FUNCTION alg_g_a_X2: LREAL
{ S7_Optimized_Access := 'true' }
    VAR_INPUT
        state: STATE;
    END_VAR

BEGIN
    alg_g_a_X2 := state.curTime;
END_FUNCTION
